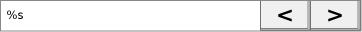
VISUALIZATION V_LoggerFilterLine  // 362x32
VAR_IN_OUT
	IOszTxtActual : STRING(80);
	IOszTxtLine : STRING(80);
END_VAR
    Rectangle (0,0 260x30), "%s", text variable: IOszTxtLine
        OnMouseClick: write the text variable via Default
    Button (260,0 50x30), "<"
        OnMouseClick: execute { IOszTxtLine := IOszTxtActual; }
    Button (310,0 50x30), ">"
        OnMouseClick: execute { IOszTxtActual := IOszTxtLine; }
END_VISUALIZATION

(* stored: Version 1.1.0.1, ProductVersion 3.1.4018.10
   Visu V_LoggerFilterLine: Id {fe1653bd-1779-44a1-a57c-2545d9c51230} *)
